Staubli VAL3: start.pgx

program start()
  local num l_nElement
begin

  sInput[0] = "forward 9"
  sInput[1] = "forward 9 gtgt"
  sInput[2] = " 1878"

  call splitString(sInput, " ", lResult)

  call splitWord(sInput, lResult)

  call trimString(sInput, sResult)

  call toUppercase(sInput[1], sResult)

  call replacePattern(sInput, "r", "HGT", sResult)

  ? "## test sub: sub(sInput, 2,4,sResult)"
  call subString(sInput, 2,10,sResult)
  call utils:printStr(sResult)

   ? "## test sub: removeString(sInput, 2,3,sResult)"
  call removeString(sInput, 2,3,sResult)
  call utils:printStr(sResult)
end
